% RSLogix 500 project LAB 2 Q4 ROBO_BAK000.RSS, saved by version 8.40.00.08 %
PROJECT "UNTITLED"    % processor: type code 162 %

PROGRAM FILES
  LAD 2   9 rungs

DATA FILES
  S2 STATUS  83 elements
  B3 BINARY  1 elements
  T4 TIMER  1 elements
  C5 COUNTER  1 elements
  R6 CONTROL  1 elements
  N7 INTEGER  1 elements
  F8 FLOAT  1 elements

LADDER 2
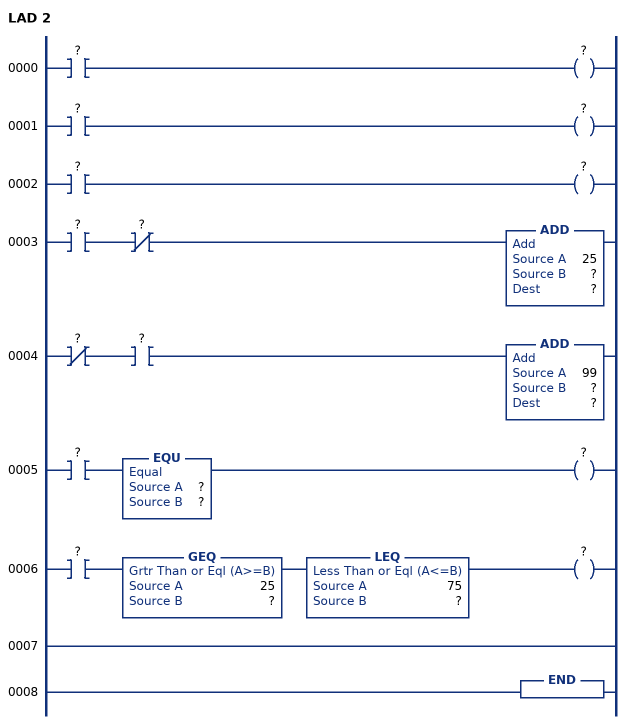
% Rung: 0 %  % edit flag set %
SOR XIC ? OTE ? EOR
% Rung: 1 %  % edit flag set %
SOR XIC ? OTE ? EOR
% Rung: 2 %  % edit flag set %
SOR XIC ? OTE ? EOR
% Rung: 3 %  % edit flag set %
SOR XIC ? XIO ? ADD 25 ? ? EOR
% Rung: 4 %  % edit flag set %
SOR XIO ? XIC ? ADD 99 ? ? EOR
% Rung: 5 %  % edit flag set %
SOR XIC ? EQU ? ? OTE ? EOR
% Rung: 6 %  % edit flag set %
SOR XIC ? GEQ 25 ? LEQ 75 ? OTE ? EOR
% Rung: 7 %  % edit flag set %
SOR EOR
% Rung: 8 %
SOR END EOR
